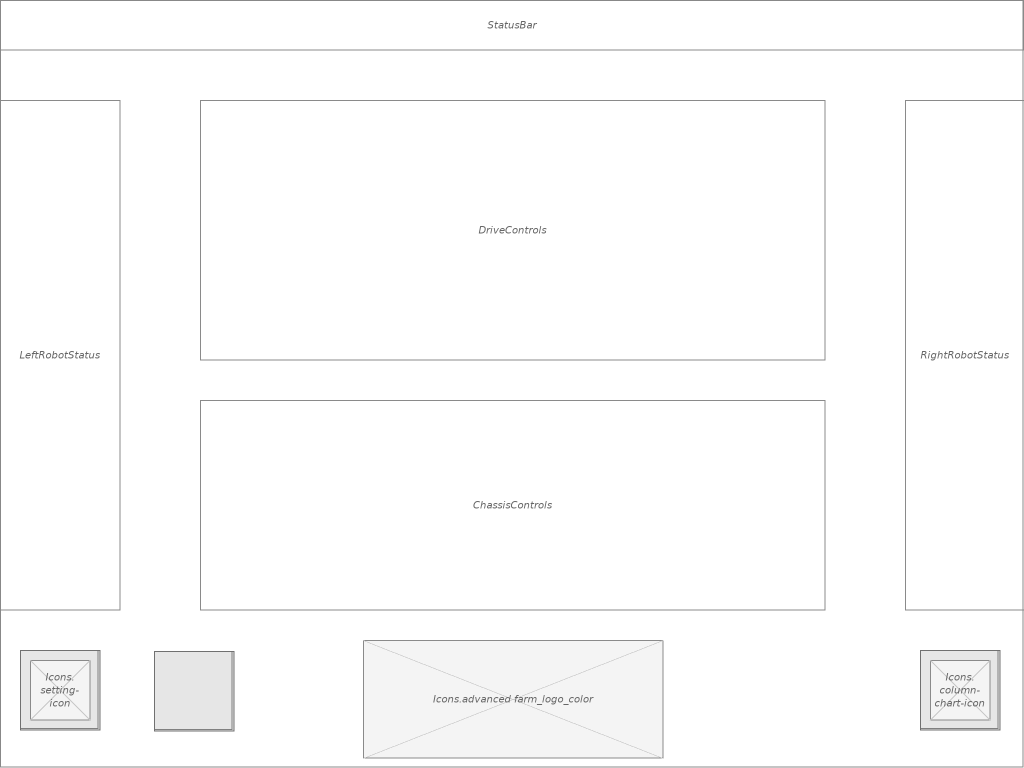
VISUALIZATION Home_Screen  // 1024x768
    Rectangle (905,100 120x510)
    Rectangle (0,100 120x510)
    Rectangle (200,400 625x210)
    Rectangle (200,100 625x260)
    Rectangle (0,0 1024x50)
    Frame (0,0 1024x50)
        shows StatusBar()
    Image (363,640 300x118), image: Icons.advanced farm_logo_color
    Group (20,650 80x80)
        OnMouseClick: change screen: Supervisor_Screen
        Button (0,0 80x80)
        Image (10,10 60x60), image: Icons.setting-icon
    Group (920,650 80x80)
        OnMouseClick: change screen: Stats_Screen
        Button (0,0 80x80)
        Image (10,10 60x60), image: Icons.column-chart-icon
    Frame (200,400 625x210), frame switch variable: UI.FrameSelector.SelectedFrame
        shows ChassisControls()
        shows RobotStatusPopup()
    Frame (200,100 625x260)
        shows DriveControls()
    Frame (0,100 120x510)
        shows LeftRobotStatus()
    Frame (905,100 120x510)
        shows RightRobotStatus()
    Button (154,651 80x80)
END_VISUALIZATION

(* stored: Version 1.1.0.1, ProductVersion 3.1.4024.15
   Visu Home_Screen: Id {f5090422-d861-4e58-8160-c3ab4d9a9b63} *)
